PROGRAM MAIN
VAR
END_VAR

END_PROGRAM

(* stored: Version 1.1.0.1
   POU MAIN: Id {54ede477-90d7-49d4-b8d4-ec990f22c660} *)
